{attribute 'qualified_only'}
{attribute 'strict'}
TYPE E_PCMControlMode :
(
	coolingMode := 0, 
	pumpMode := 1
);
END_TYPE

(* stored: Version 1.1.0.1, ProductVersion 3.1.4024.10
   DUT E_PCMControlMode: Id {019932c9-8690-45af-a63c-bc8b58feb7c5} *)
